INTERFACE I_LinearDrive EXTENDS I_Drive

{attribute 'monitoring':='call'}
PROPERTY AtHome : BOOL
GET
END_GET
END_PROPERTY

{attribute 'monitoring':='call'}
PROPERTY HomeSet : BOOL
GET
END_GET
END_PROPERTY

METHOD homingSequence : BOOL
VAR_INPUT
END_VAR
END_METHOD

METHOD toHome : BOOL
VAR_INPUT
END_VAR
END_METHOD

END_INTERFACE

(* stored: Version 1.1.0.1, ProductVersion 3.1.4024.11
   Itf I_LinearDrive: Id {5de96b94-292d-466c-b578-4a59d3d49d3e}
   Property AtHome: Id {02e0ea02-9ef6-49be-96cc-76eb527fd724}
   Get Get: Id {426cb164-5327-41c5-9468-31545729bac1}
   Property HomeSet: Id {de35e24c-c52f-494a-a4e0-97a9c626e3b7}
   Get Get: Id {b96a860e-a293-49cc-ae54-1bf75e93fa20}
   Method homingSequence: Id {32bc7dae-a9cd-4699-b94e-c6fc22643c52}
   Method toHome: Id {d087b628-9fa2-4cc9-8120-262adf273af5} *)
